SUBAPPLICATION AX_TO_QXA_BG_PUBLISH (* Treibt aus einem bereits fertigen AX-Zustand (z.B. per OR mehrerer Quellen zusammengefuehrt - gestaffeltes Gruppensignal, Einzel-Toggle, IO-Diag-Testbutton) 1 physischen Ausgang + Hintergrundfarbe (SoftKey+AUX) + lokalen State-Publish (Web-Client/OPC-Dashboard). Gegenstueck zu MyLib::sys::AX_SoftkeyToggle_RS_TO_QXA_BG (das den Toggle/Reset noch selbst erzeugt) - hier liegt der AX-Zustand bereits fertig vor und muss nur noch auf Ausgang+Hintergrund+Publish verteilt werden. *)
  (* Standard: 61499-2; Description: Copyright (c) 2026 Meisterschulen am Ostbahnhof This program and the accompanying materials are made available under the terms of the Eclipse Public License 2.0 which is available at https://www.eclipse.org/legal/epl-2.0/ SPDX-License-Identifier: EPL-2.0 *)
  (* Version 1.0, 2026-09-15, Franz Höpfinger, Meisterschulen am Ostbahnhof, initial implementation - aus Baender_EinAus.SUB herausgeloest (AX_SPLIT_2_Igel/_Elevator/_Querband + DigitalOutput_Igel/_Elevator/_Querband + GreenWhiteBackground_Igel/_Elevator/_Querband, 3x identisch). ID_STATE_WRITE neu ergaenzt (Franz: Web-Mirror braucht fuer die Einzel-Baender-Softkeys einen eigenen State-Publish, bisher nirgends vorhanden). *)
  PACKAGE MyLib::sys;
  IMPORT isobus::UT::Q::const::IDs::ID_NULL;
  IMPORT logiBUS::io::DQ::logiBUS_DO;
  IMPORT logiBUS::io::DQ::logiBUS_DO_S;
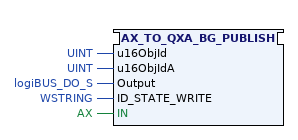
  VAR_INPUT
    u16ObjId : UINT := ID_NULL; (* Object ID Softkey - traegt die Hintergrundfarbe *)
    u16ObjIdA : UINT := ID_NULL; (* Object ID AuxFunction2 (Joystick) - zeigt Hintergrundfarbe am Aux-Handle mit *)
    Output : logiBUS::io::DQ::logiBUS_DO_S := logiBUS_DO::Invalid; (* Identify the Output Output_Q1..Q12 *)
    ID_STATE_WRITE : WSTRING; (* Lokale Publish-Adresse (ACTION=WRITE) fuer den tatsaechlichen Zustand - wird von Web-Client/Dashboard remote abonniert *)
  END_VAR
  SOCKETS
    IN : adapter::types::unidirectional::AX; (* Fertiger AX-Zustand (bereits zusammengefuehrt) - wird auf Ausgang+Hintergrund+Publish verteilt *)
  END_SOCKETS
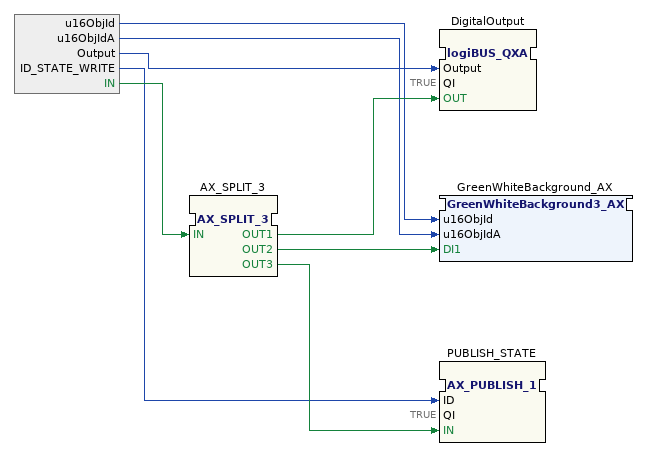
  FBS
    AX_SPLIT_3 : adapter::events::unidirectional::AX_SPLIT_3;
    DigitalOutput : logiBUS::io::DQ::logiBUS_QXA(QI := TRUE);
    PUBLISH_STATE : adapter::net::AX_PUBLISH_1(QI := TRUE);
  END_FBS
  SUBAPPS
    GreenWhiteBackground_AX : MyLib::sys::GreenWhiteBackground3_AX;
  END_SUBAPPS
  DATA_CONNECTIONS
    u16ObjId TO GreenWhiteBackground_AX.u16ObjId;
    u16ObjIdA TO GreenWhiteBackground_AX.u16ObjIdA;
    Output TO DigitalOutput.Output;
    ID_STATE_WRITE TO PUBLISH_STATE.ID;
  END_CONNECTIONS
  ADAPTER_CONNECTIONS
    IN TO AX_SPLIT_3.IN;
    AX_SPLIT_3.OUT1 TO DigitalOutput.OUT;
    AX_SPLIT_3.OUT2 TO GreenWhiteBackground_AX.DI1;
    AX_SPLIT_3.OUT3 TO PUBLISH_STATE.IN;
  END_CONNECTIONS
END_SUBAPPLICATION
